FUNCTION_BLOCK ABSTRACT FB_Shape
VAR
	_color : ITF_color;
END_VAR

METHOD ABSTRACT Draw : STRING
END_METHOD

METHOD FB_init : BOOL
VAR_INPUT
	bInitRetains : BOOL; // if TRUE, the retain variables are initialized (warm start / cold start)
	bInCopyCode : BOOL;  // if TRUE, the instance afterwards gets moved into the copy code (online change)
	Color : ITF_Color;
END_VAR
THIS^._color := Color;
END_METHOD

END_FUNCTION_BLOCK

(* stored: Version 1.1.0.1, ProductVersion 3.1.4024.12
   POU FB_Shape: Id {c353f373-9ede-4c31-83a9-a7197bda022a}, SpecialFunc None
   Method Draw: Id {238a75eb-020f-4c4c-9456-88d1cd5ae639}
   Method FB_init: Id {42591783-ae3d-48ef-8d1f-58b95c90d4c2} *)
